ABB RobotStudio station: RobotStudio.rsstn

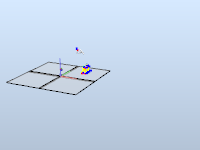
Station RobotStudio (saved by RobotStudio 22.1.9826.0)
Controller IRB140_6_81_1
  mechanical unit ROB_1: IRB140_6_81_C_03, 6 joints, base frame (0, 0, 0) mm
Layout (positions relative to the parent item):
  - IRB140_6_81_C_03 [mechanism, from Robots\IRB140_6_81_C_G_03.rslib] at (0, 0, 0) mm; joint values [0, 0, 0, 0, 0, 0] (rad or m)
  - Marcador [mechanism, from Lab1\Marcador.rslib] at (515, 0, 712) mm, rotated rx 0 ry 90 rz 0 deg
  - Frame_2 [frame] at (31.27, 0, 208.36) mm, rotated rx 180 ry 0 rz 180 deg
Attachment: Marcador is attached to IRB140_6_81_C_03 / Link6
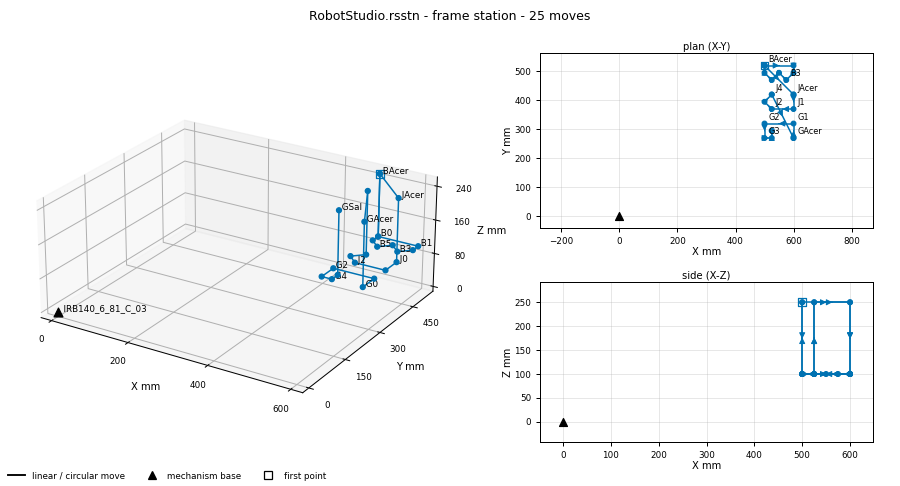
[picture p0: tool path of RobotStudio.rsstn in frame station, 25 of 27 moves have a stored position in this frame; points joined in program order, loops and branches not executed]
Targets, tools, work objects and paths stored in the station, written as RAPID:
! task T_ROB1
MODULE CalibData
  PERS tooldata TMarcador:=[TRUE,[[31.268,0,208.361],[0.923879533,0,-0.382683432,0]],[0.168,[-21.829,0,103.099],[1,0,0,0],0,0,0]];
  TASK PERS wobjdata Tablero:=[FALSE,TRUE,"",[[500,520,100],[0.707106781,0,0.707106781,0]],[[0,0,0],[1,0,0,0]]];
ENDMODULE

! task T_ROB1
MODULE Module1
  CONST robtarget B0:=[[0,0,0],[1,0,0,0],[0,0,0,0],[9E+09,9E+09,9E+09,9E+09,9E+09,9E+09]];
  CONST robtarget B1:=[[0,0,100],[1,0,0,0],[0,-1,1,0],[9E+09,9E+09,9E+09,9E+09,9E+09,9E+09]];
  CONST robtarget B2:=[[0,-25,100],[1,0,0,0],[0,-1,1,0],[9E+09,9E+09,9E+09,9E+09,9E+09,9E+09]];
  CONST robtarget B3:=[[0,-50,75],[1,0,0,0],[0,-1,1,0],[9E+09,9E+09,9E+09,9E+09,9E+09,9E+09]];
  CONST robtarget B4:=[[0,-25,50],[1,0,0,0],[0,-1,1,0],[9E+09,9E+09,9E+09,9E+09,9E+09,9E+09]];
  CONST robtarget B5:=[[0,-50,25],[1,0,0,0],[0,-2,1,0],[9E+09,9E+09,9E+09,9E+09,9E+09,9E+09]];
  CONST robtarget B6:=[[0,-25,0],[1,0,0,0],[0,-1,1,0],[9E+09,9E+09,9E+09,9E+09,9E+09,9E+09]];
  CONST robtarget BAcer:=[[-150,0,0],[1,0,0,0],[0,-1,1,0],[9E+09,9E+09,9E+09,9E+09,9E+09,9E+09]];
  CONST robtarget J0:=[[0,-100,100],[1,0,0,0],[0,-2,1,0],[9E+09,9E+09,9E+09,9E+09,9E+09,9E+09]];
  CONST robtarget J1:=[[0,-150,100],[1,0,0,0],[0,-2,1,0],[9E+09,9E+09,9E+09,9E+09,9E+09,9E+09]];
  CONST robtarget J2:=[[0,-150,25],[1,0,0,0],[0,-2,1,0],[9E+09,9E+09,9E+09,9E+09,9E+09,9E+09]];
  CONST robtarget J3:=[[0,-125,0],[1,0,0,0],[0,-2,1,0],[9E+09,9E+09,9E+09,9E+09,9E+09,9E+09]];
  CONST robtarget J4:=[[0,-100,25],[1,0,0,0],[0,-2,1,0],[9E+09,9E+09,9E+09,9E+09,9E+09,9E+09]];
  CONST robtarget G0:=[[0,-250,100],[1,0,0,0],[0,-2,1,0],[9E+09,9E+09,9E+09,9E+09,9E+09,9E+09]];
  CONST robtarget G1:=[[0,-200,100],[1,0,0,0],[0,-2,1,0],[9E+09,9E+09,9E+09,9E+09,9E+09,9E+09]];
  CONST robtarget G2:=[[0,-200,0],[1,0,0,0],[0,-2,1,0],[9E+09,9E+09,9E+09,9E+09,9E+09,9E+09]];
  CONST robtarget G3:=[[0,-250,0],[1,0,0,0],[0,-2,1,0],[9E+09,9E+09,9E+09,9E+09,9E+09,9E+09]];
  CONST robtarget G4:=[[0,-250,25],[1,0,0,0],[0,-2,1,0],[9E+09,9E+09,9E+09,9E+09,9E+09,9E+09]];
  CONST robtarget G5:=[[0,-225,25],[1,0,0,0],[0,-2,1,0],[9E+09,9E+09,9E+09,9E+09,9E+09,9E+09]];
  CONST robtarget JAcer:=[[-150,-100,100],[1,0,0,0],[0,-1,1,0],[9E+09,9E+09,9E+09,9E+09,9E+09,9E+09]];
  CONST robtarget GAcer:=[[-150,-250,100],[1,0,0,0],[0,-2,1,0],[9E+09,9E+09,9E+09,9E+09,9E+09,9E+09]];
  CONST robtarget JSal_10:=[[-150,-100,25],[1,0,0,0],[0,-1,1,0],[9E+09,9E+09,9E+09,9E+09,9E+09,9E+09]];
  CONST robtarget GSal:=[[-150,-225,25],[1,0,0,0],[0,-2,1,0],[9E+09,9E+09,9E+09,9E+09,9E+09,9E+09]];
  CONST robtarget HOMEP_10:=[[-679.5,-520,6.29],[0.707106781,0,-0.707106781,0],[0,-2,-2,0],[9E+09,9E+09,9E+09,9E+09,9E+09,9E+09]];
  CONST jointtarget HOME:=[[0,0,0,0,0,0],[9E+09,9E+09,9E+09,9E+09,9E+09,9E+09]];
  CONST jointtarget Intermedio:=[[39.820347786,7.402611956,17.639279428,-47.788627471,37.688106161,71.623214618],[9E+09,9E+09,9E+09,9E+09,9E+09,9E+09]];
  PROC AcerYLetras()
    MoveL BAcer,v1000,z100,TMarcador\WObj:=Tablero;
    MoveL B0,v1000,z100,TMarcador\WObj:=Tablero;
    MoveL B1,v1000,z100,TMarcador\WObj:=Tablero;
    MoveL B2,v1000,z100,TMarcador\WObj:=Tablero;
    MoveL B3,v1000,z100,TMarcador\WObj:=Tablero;
    MoveL B4,v1000,z100,TMarcador\WObj:=Tablero;
    MoveL B5,v1000,z100,TMarcador\WObj:=Tablero;
    MoveL B6,v1000,z100,TMarcador\WObj:=Tablero;
    MoveL B0,v1000,z100,TMarcador\WObj:=Tablero;
    MoveL BAcer,v1000,z100,TMarcador\WObj:=Tablero;
    MoveL JAcer,v1000,z100,TMarcador\WObj:=Tablero;
    MoveL J0,v1000,z100,TMarcador\WObj:=Tablero;
    MoveL J1,v1000,z100,TMarcador\WObj:=Tablero;
    MoveL J2,v1000,z100,TMarcador\WObj:=Tablero;
    MoveL J3,v1000,z100,TMarcador\WObj:=Tablero;
    MoveL J4,v1000,z100,TMarcador\WObj:=Tablero;
    MoveL JSal_10,v1000,z100,TMarcador\WObj:=Tablero;
    MoveL GAcer,v1000,z100,TMarcador\WObj:=Tablero;
    MoveL G0,v1000,z100,TMarcador\WObj:=Tablero;
    MoveL G1,v1000,z100,TMarcador\WObj:=Tablero;
    MoveL G2,v1000,z100,TMarcador\WObj:=Tablero;
    MoveL G3,v1000,z100,TMarcador\WObj:=Tablero;
    MoveL G4,v1000,z100,TMarcador\WObj:=Tablero;
    MoveL G5,v1000,z100,TMarcador\WObj:=Tablero;
    MoveL GSal,v1000,z100,TMarcador\WObj:=Tablero;
  ENDPROC
  PROC HomeP()
    MoveAbsJ HOME,v1000,z100,TMarcador\WObj:=Tablero;
  ENDPROC
  PROC AcerInter()
    MoveAbsJ Intermedio,v1000,z100,TMarcador\WObj:=Tablero;
  ENDPROC
ENDMODULE

